DATA_BLOCK "Test"
{ S7_Optimized_Access := 'FALSE' }
VERSION : 0.1
NON_RETAIN
   STRUCT
      Member1 : Struct
         Member2 : Struct
            Member3 : Struct
               Member4 : Struct
                  Member5 : Array[0..1] of Bool;
               END_STRUCT;
            END_STRUCT;
         END_STRUCT;
         Member21 : Int;
      END_STRUCT;
      Member12 : Array[0..1] of String[32];
   END_STRUCT;


BEGIN

END_DATA_BLOCK

